Universal Robots PolyScope program: Start Heating Welder.urp

Program Start Heating Welder (installation=default directory=/programs/UPF createdIn=5.14.5 lastSavedIn=5.14.5 robotSerialNumber=20236801216)
Calibrated DH parameters: a=[-0.000021, -0.748897, -0.28186, -0.00004, -0.000055, 0]; d=[0.236225, -424.082933, -1564.66872, 1988.95162, 0.159094, 0.153873]; alpha=[1.570844, 0.001002, 0.000337, 1.571488, -1.569996, 0]; deltaTheta=[0, -0.516316, 5.626292, 1.173211, 0.000001, 0]
InitVariablesNode
Robot Program (runOnlyOnce=true)
  HwResp := [0,0,0]
  SuppressedNode
    junk := [0,0,0]
  URCap WireTank Serial (WireTank Serial, WireTank, LLC) dataModel(Command=[252,72,49], NODE_TITLE=Serial Bridge uH1, QUERY=true, byte_array=true, OUTPUT_ENTRY=Static, Variable(key=OUTPUT_VARIABLE, variable=junk))
  URCap WireTank Serial (WireTank Serial, WireTank, LLC) dataModel(Command=[252,72,49], NODE_TITLE=Serial Bridge uH1, QUERY=true, byte_array=true, OUTPUT_ENTRY=Static, Variable(key=OUTPUT_VARIABLE, variable=HwResp))
  SuppressedNode
    Wait Sleep waitTime=5
  SuppressedNode
    Popup Message (haltProgram=false message=heating started. push to stop inputType=Text)
  SuppressedNode
    URCap WireTank Serial (WireTank Serial, WireTank, LLC) dataModel(NODE_TITLE=Serial Bridge uh?, byte_array=true, Command=[252,104,63], OUTPUT_ENTRY=Static, QUERY=true, Variable(key=OUTPUT_VARIABLE, variable=HwResp))
  SuppressedNode
    Popup Message (haltProgram=false inputType=Variable) variable=HwResp
  SuppressedNode
    Wait Sleep waitTime=20
  SuppressedNode
    URCap WireTank Serial (WireTank Serial, WireTank, LLC) dataModel(byte_array=true, Command=[252,72,48], NODE_TITLE=Serial Bridge uH0, QUERY=false, OUTPUT_ENTRY=Static, Variable(key=OUTPUT_VARIABLE, variable=HwResp))
  SuppressedNode
    Popup Message (haltProgram=false message=heating stopped. push to start inputType=Text)
  'set the temp reader to high voltage (off) when program is running and low volt (on) when program not running'
  Script: set_runstate_standard_digital_output_to_value(2,3)
  'set 5V power to munsch powerbox to high (on) when a program is started and low on unscheduled stop'
  Script: set_runstate_standard_digital_output_to_value(1,5)
